Fanuc TP program (LS listing): SYNC2WAIT.LS

/PROG  SYNC2WAIT
/ATTR
OWNER		= MNEDITOR;
COMMENT		= "";
PROG_SIZE	= 278;
CREATE		= DATE 11-05-20  TIME 11:03:02;
MODIFIED	= DATE 11-06-15  TIME 17:54:20;
FILE_NAME	= SYNC2WAI;
VERSION		= 0;
LINE_COUNT	= 3;
MEMORY_SIZE	= 646;
PROTECT		= READ;
TCD:  STACK_SIZE	= 0,
      TASK_PRIORITY	= 50,
      TIME_SLICE	= 0,
      BUSY_LAMP_OFF	= 0,
      ABORT_REQUEST	= 0,
      PAUSE_REQUEST	= 0;
DEFAULT_GROUP	= *,*,*,*,*;
CONTROL_CODE	= 00000000 00000000;
/APPL
  SPOT : TRUE ;
/MN
   1:  CALL MSYNC(1,16,16,9999999,16,9999999,16,9999999,16,9999999) ;
   2:   ;
   3:   ;
/POS
/END
